Universal Robots PolyScope program: tcpip_comm_v2.urp

Program tcpip_comm_v2 (installation=comm directory=/programs/usbdisk/RobotControl createdIn=5.11.9 lastSavedIn=5.14.5 robotSerialNumber=20225501312)
Calibrated DH parameters: a=[0.000177, -0.405867, -0.359302, -0.000009, 0.00008, 0]; d=[0.162556, -59.259033, 22.634856, 36.757695, 0.099775, 0.099535]; alpha=[1.570983, 0.00214, 0.004319, 1.570342, -1.569638, 0]; deltaTheta=[0, -0.302866, 6.171309, 0.414749, 0.000002, -0.000001]
InitVariablesNode
BeforeStart
  open_socket := socket_open("192.168.65.197",8888,"ur5e_pc")
  Loop While (checkContinuously=false) expression=open_socket≟ False
    open_socket := socket_open("192.168.65.197",8888,"ur5e_pc")
Robot Program (runOnlyOnce=false)
  SuppressedNode
    MoveJ speed 60 deg/s, acceleration 80 deg/s^2 (useActiveTCP=true) feature=Base
      Waypoint Waypoint_1: TCP in base x=580.549 y=-78.899 z=424.087 mm, rx=-2.1574 ry=2.2822 rz=0.0245 rad; joints [4.983, -104.184, -56.406, -109.948, 90.735, 8.274] deg; TCP offset x=0 y=0 z=180.13 mm, rx=0 ry=0 rz=0 rad
  If open_socket≟ True
    Folder string
      'read string'
      str := socket_read_string("ur5e_pc")
      Loop While (checkContinuously=false) expression=str≟""
        str := socket_read_string("ur5e_pc")
        Wait Sleep waitTime=0.01
      'send string'
      was_send := socket_send_string("ACK","ur5e_pc")
      Loop While (checkContinuously=false) expression=was_send≟ False
        was_send := socket_send_string("ACK","ur5e_pc")
        Wait Sleep waitTime=0.01
      Wait Sleep waitTime=0.01
    Folder integer
      'read int'
      data := socket_read_binary_integer(1,"ur5e_pc")
      Loop While (checkContinuously=false) expression=data[0]≟0
        data := socket_read_binary_integer(1,"ur5e_pc")
        Wait Sleep waitTime=0.01
      'send int'
      was_send := socket_send_int(9,"ur5e_pc")
      Loop While (checkContinuously=false) expression=was_send≟ False
        was_send := socket_send_int(9,"ur5e_pc")
        Wait Sleep waitTime=0.01
      Wait Sleep waitTime=0.01
    Folder integer array
      'read Int array'
      array_size := 3
      data3 := socket_read_binary_integer(array_size,"ur5e_pc")
      Loop While (checkContinuously=false) expression=data3[0]≟0
        data3 := socket_read_binary_integer(array_size,"ur5e_pc")
        Wait Sleep waitTime=0.01
      'send int array'
      int_array := [4, 5, 6]
      str_int := to_str(int_array)
      was_send := socket_send_string(str_int,"ur5e_pc")
      Loop While (checkContinuously=false) expression=was_send≟ False
        was_send := socket_send_string(str_int,"ur5e_pc")
        Wait Sleep waitTime=0.01
      Wait Sleep waitTime=0.01
    Folder float
      'get one float'
      data4 := socket_read_ascii_float(1,"ur5e_pc")
      Loop While (checkContinuously=false) expression=data4[0]≟0
        data4 := socket_read_ascii_float(1,"ur5e_pc")
        Wait Sleep waitTime=0.01
      'send array of floats'
      send_floats := 8.8
      str_floats := to_str(send_floats)
      was_send := socket_send_string(str_floats,"ur5e_pc")
      Loop While (checkContinuously=false) expression=was_send≟ False
        was_send := socket_send_string(str_floats,"ur5e_pc")
        Wait Sleep waitTime=0.01
    Folder float array
      'get array of floats'
      data2 := socket_read_ascii_float(3,"ur5e_pc")
      Loop While (checkContinuously=false) expression=data2[0]≟0
        data2 := socket_read_ascii_float(3,"ur5e_pc")
        Wait Sleep waitTime=0.01
      'send array of floats'
      send_floats2 := [4.4, 5.5, 6.6]
      str_floats := to_str(send_floats2)
      was_send := socket_send_string(str_floats,"ur5e_pc")
      Loop While (checkContinuously=false) expression=was_send≟ False
        was_send := socket_send_string(str_floats,"ur5e_pc")
        Wait Sleep waitTime=0.01
    Script: socket_close("ur5e_pc")
    Halt
